// TIA Portal V16 export
// export: Created 2025-12-18T09:30:40.4208466Z, ExportSetting WithDefaults, DisplayName Totally Integrated Automation Portal, DisplayVersion V16, DisplayName TIA Portal Version Control Interface, DisplayVersion V16, DisplayName TIA Portal Openness, DisplayVersion V16, DisplayName STEP 7 Professional, DisplayVersion V16, DisplayName STEP 7 Safety, DisplayVersion V16, DisplayName WinCC Advanced, DisplayVersion V16
FUNCTION_BLOCK "Sequence Data Management"   // FB3, LAD
{ S7_Optimized_Access := 'TRUE' }
VERSION : 0.1
// stored: AutoNumber true, IsIECCheckEnabled false, IsRetainMemResEnabled false, MemoryReserve 100, SetENOAutomatically false, UDAEnableTagReadback false
   VAR
      WorkStationList1 : Array[0..9] of DInt;
      WorkStationList2 : Array[0..9] of DInt;
      WorkStationList3 : Array[0..9] of DInt;
   END_VAR
   // WorkStationList1[0..9] := -1;
   // WorkStationList2[0..9] := -1;
   // WorkStationList3[0..9] := -1;
   VAR_TEMP   // added for the SCL form of the ladder/FBD networks
      _w1 : Bool;
      _w2 : Bool;
   END_VAR
BEGIN

REGION Network 1
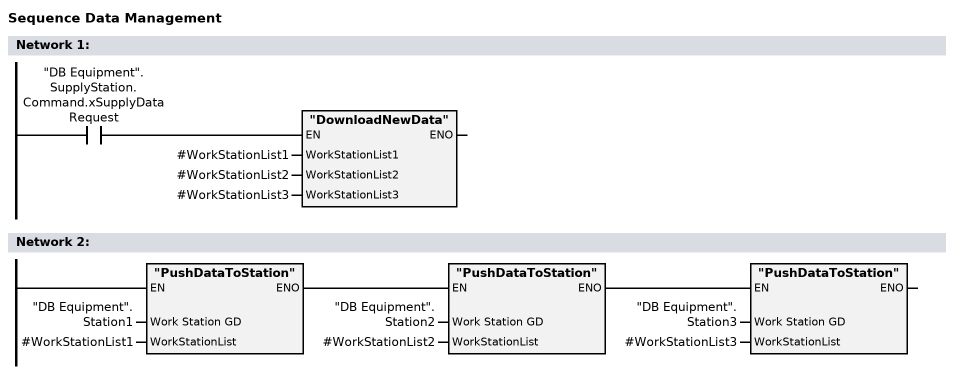
   RUNG wire#powerrail
      Contact( "DB Equipment".SupplyStation.Command.xSupplyDataRequest )
      "DownloadNewData"(WorkStationList1 := #WorkStationList1, WorkStationList2 := #WorkStationList2, WorkStationList3 := #WorkStationList3)
   END_RUNG
   // the same network as SCL:
   IF "DB Equipment".SupplyStation.Command.xSupplyDataRequest THEN
       "DownloadNewData"(WorkStationList1 := #WorkStationList1,
                         WorkStationList2 := #WorkStationList2,
                         WorkStationList3 := #WorkStationList3);
   END_IF;
END_REGION

REGION Network 2
   RUNG wire#powerrail
      "PushDataToStation"("Work Station GD" := "DB Equipment".Station1, WorkStationList := #WorkStationList1)
      "PushDataToStation"("Work Station GD" := "DB Equipment".Station2, WorkStationList := #WorkStationList2)
      "PushDataToStation"("Work Station GD" := "DB Equipment".Station3, WorkStationList := #WorkStationList3)
   END_RUNG
   // the same network as SCL:
   "PushDataToStation"("Work Station GD" := "DB Equipment".Station1,
                       WorkStationList := #WorkStationList1,
                       ENO => #_w1);
   "PushDataToStation"(EN := #_w1,
                       "Work Station GD" := "DB Equipment".Station2,
                       WorkStationList := #WorkStationList2,
                       ENO => #_w2);
   IF #_w2 THEN
       "PushDataToStation"("Work Station GD" := "DB Equipment".Station3, WorkStationList := #WorkStationList3);
   END_IF;
END_REGION
END_FUNCTION_BLOCK
